Fanuc KAREL source: kt00190.KL

-- PROVISIONAL review KL for V940-1; original PC SHA256 2b2267b0035dd17bde1c925842c018e2dd0487f37fa7a3874e19392c912d02e0
-- Incomplete behavior may be omitted. Consult companion uncertainty JSON. Do not deploy.
PROGRAM KT00190
%NOLOCKGROUP
VAR
  OUT : REAL
-- UNRESOLVED_DECL H1 type=002017
-- UNRESOLVED_DECL Y2 type=002018
BEGIN
  -- V9_ZERO_TABLE_METADATA_HINT layout=0001; no indexed target words; source/name/runtime held
  -- UNRESOLVED_PC offsets 5-19; opcodes 2E,22,9D,33,B4
  -- UNRESOLVED_PC offsets 24-38; opcodes 2E,22,9D,33,B2
  -- UNRESOLVED_PC offsets 43-69; opcodes 22,9D,33,B3,22,9D,33,B1,56,64,23
  -- UNRESOLVED_PC offsets 74-78; opcodes 7F
END KT00190
